(* CODESYS project device_plc_f5a.project

Project tree, tasks and I/O mapping:
  Device : C6 SMART BASIC, KEB - Karl E. Brinkmann GmbH, version 3.5.6.41
    application Application
      libraries: Standard, * (System); KEB_Gateway_Utility, * (KEB - Karl E. Brinkmann GmbH); SysTimeCore, * (System); CmpErrors, * (System); SysSocket, * (System); KEB_Drive_Utility, * (KEB - Karl E. Brinkmann GmbH); KEB_Base, * (KEB - Karl E. Brinkmann GmbH); CmpEventMgr, 3.5.5.0 (System); Component Manager, 3.5.5.0 (System); CmpApp, 3.5.6.0 (System); CmpIecTask, 3.5.5.0 (System)
      task MainTask (cyclic, interval t#4ms, priority 0) calls PLC_PRG, Gateway
      task EtherCAT_Master_C6_SMART (externalevent, external event EVENT_ECM_DC, priority 0) calls EtherCAT_Master_C6_SMART.EtherCAT_Task [EtherCAT_Master_C6_SMART.EtherCAT_Task]
      program PLC_PRG [ST]: ErrorHandling
      program MAIN [ST]
      Gateway/
        program Gateway [FBD]
        global variables GVL_GATEWAY
        global variables GVL_APP
        program SampleReadDriveParameter [FBD]
        program SampleReadMultipleParameter [ST]
        program SampleWriteDriveParameter [ST]
      SDO_RW/
        program ReadParameters [ST]
        FB/
          function block ReadPara [ST]
          function block WritePara [ST]: Dint_ToArrayOfByte
          function ArrayOfByte_to_Dword [ST]
          function block ReadParaEdge [ST]
      TCP_Server/
        function block SocketComm [ST]
        program ServerSocket [ST]: SplitRxBuffer, InitSocketFB, ComposeTxBuffer
        program PrepareStopFunction [ST]
        global variables GVL_TCP
    EtherCAT_Master_C6_SMART : EtherCAT Master C6 SMART, KEB - Karl E. Brinkmann GmbH, version 3.5.5.0
      KEB_C6_SMART_Coupler : KEB_C6_SMART_Coupler (3A E-Bus), KEB - Karl E. Brinkmann GmbH, version Revision=16#00000003
          settings: DC sync0 cycletime = 8000; DC sync1 cycletime = 8000
      KEB_F5_generic_MDP_ : KEB_F5_generic (MDP), KEB - Karl E. Brinkmann GmbH, version Revision=16#00000000
          settings: Number of Outputs = 3; Number of Inputs = 3; Number of Infos about Outputs = 3; Number of Infos about Inputs = 3; EnableExpertSettings = True; Sync.Length = 8; Sync.Length = 8; FMMU.Length = 8; FMMU.Length = 8; Number of RxPDOs of the Slave = 1; Number of TxPDOs of the Slave = 1; DC sync0 cycletime = 8000; DC enable = 1; DC sync0 enable = 1; DC sync0 factor = 'x 1'; DC sync0 shift time = 0; DC sync1 cycletime = 8000; DC sync1 enable = 0; DC sync1 factor = 'x 1'; DC sync1 shift time = 0; DCSetting = 1; RxTxPdo.NumberofExcludes = 0; RxTxPdo.NumberofEntries = 3; RxTxPdo.Index = 16#1600; RxTxPdo.Fixed = False; RxTxPdo.Mandatory = False; RxTxPdo.Virtual = False; RxTxPdo.Sm = 2; RxTxPdo.Su = 0; RxTxPdo.Name = 'Outputs'; RxTxPdo.DependOnSlot = True; RxTxPdo.DependOnSlotGroup = False; std_PD_map_F5_ PS34: ctm position [0x3322.0].Index = 16#3322; std_PD_map_F5_ PS34: ctm position [0x3322.0].SubIndex = 1; std_PD_map_F5_ PS34: ctm position [0x3322.0].Size = 32; std_PD_map_F5_ PS34: ctm position [0x3322.0].Offset = 0; std_PD_map_F5_ PS34: ctm position [0x3322.0].DependOnSlot = False; std_PD_map_F5_ PS34: ctm position [0x3322.0].DependOnSlotGroup = False; std_PD_map_F5_ Sy52: set speed value [0x2034.0].Index = 16#2034; std_PD_map_F5_ Sy52: set speed value [0x2034.0].SubIndex = 1;
            std_PD_map_F5_ Sy52: set speed value [0x2034.0].Size = 16; std_PD_map_F5_ Sy52: set speed value [0x2034.0].Offset = 0; std_PD_map_F5_ Sy52: set speed value [0x2034.0].DependOnSlot = False; std_PD_map_F5_ Sy52: set speed value [0x2034.0].DependOnSlotGroup = False; std_PD_map_F5_ Sy50: control word (low) [0x2032.0].Index = 16#2032; std_PD_map_F5_ Sy50: control word (low) [0x2032.0].SubIndex = 1; std_PD_map_F5_ Sy50: control word (low) [0x2032.0].Size = 16; std_PD_map_F5_ Sy50: control word (low) [0x2032.0].Offset = 0; std_PD_map_F5_ Sy50: control word (low) [0x2032.0].DependOnSlot = False; std_PD_map_F5_ Sy50: control word (low) [0x2032.0].DependOnSlotGroup = False; RxTxPdo.NumberofExcludes = 0; RxTxPdo.NumberofEntries = 3; RxTxPdo.Index = 16#1A00; RxTxPdo.Fixed = False; RxTxPdo.Mandatory = False; RxTxPdo.Virtual = False; RxTxPdo.Sm = 3; RxTxPdo.Su = 0; RxTxPdo.Name = 'Inputs'; RxTxPdo.DependOnSlot = True; RxTxPdo.DependOnSlotGroup = False; std_PD_map_F5_ ru54: actual position [0x2236.0].Index = 16#2236; std_PD_map_F5_ ru54: actual position [0x2236.0].SubIndex = 1; std_PD_map_F5_ ru54: actual position [0x2236.0].Size = 32; std_PD_map_F5_ ru54: actual position [0x2236.0].Offset = 0; std_PD_map_F5_ ru54: actual position [0x2236.0].DependOnSlot = False; std_PD_map_F5_ ru54: actual position [0x2236.0].DependOnSlotGroup = False; std_PD_map_F5_ Sy53: actual speed value [0x2035.0].Index = 16#2035; std_PD_map_F5_ Sy53: actual speed value [0x2035.0].SubIndex = 1; std_PD_map_F5_ Sy53: actual speed value [0x2035.0].Size = 16; std_PD_map_F5_ Sy53: actual speed value [0x2035.0].Offset = 0; std_PD_map_F5_ Sy53: actual speed value [0x2035.0].DependOnSlot = False; std_PD_map_F5_ Sy53: actual speed value [0x2035.0].DependOnSlotGroup = False; std_PD_map_F5_ Sy51: status word (low) [0x2033.0].Index = 16#2033; std_PD_map_F5_ Sy51: status word (low) [0x2033.0].SubIndex = 1; std_PD_map_F5_ Sy51: status word (low) [0x2033.0].Size = 16; std_PD_map_F5_ Sy51: status word (low) [0x2033.0].Offset = 0; std_PD_map_F5_ Sy51: status word (low) [0x2033.0].DependOnSlot = False; std_PD_map_F5_ Sy51: status word (low) [0x2033.0].DependOnSlotGroup = False; std_PD_map_F5_ PS34: ctm position [0x3322.0].Name = 'std_PD_map_F5_ PS34: ctm position [0x3322.0]';
            std_PD_map_F5_ PS34: ctm position [0x3322.0].DataType = 'DINT'; std_PD_map_F5_ PS34: ctm position [0x3322.0].Default = ''; std_PD_map_F5_ PS34: ctm position [0x3322.0].Comment = ''; std_PD_map_F5_ Sy52: set speed value [0x2034.0].Name = 'std_PD_map_F5_ Sy52: set speed value [0x2034.0]'; std_PD_map_F5_ Sy52: set speed value [0x2034.0].DataType = 'INT'; std_PD_map_F5_ Sy52: set speed value [0x2034.0].Default = ''; std_PD_map_F5_ Sy52: set speed value [0x2034.0].Comment = ''; std_PD_map_F5_ Sy50: control word (low) [0x2032.0].Name = 'std_PD_map_F5_ Sy50: control word (low) [0x2032.0]'; std_PD_map_F5_ Sy50: control word (low) [0x2032.0].DataType = 'INT'; std_PD_map_F5_ Sy50: control word (low) [0x2032.0].Default = ''; std_PD_map_F5_ Sy50: control word (low) [0x2032.0].Comment = ''; std_PD_map_F5_ ru54: actual position [0x2236.0].Name = 'std_PD_map_F5_ ru54: actual position [0x2236.0]'; std_PD_map_F5_ ru54: actual position [0x2236.0].DataType = 'DINT'; std_PD_map_F5_ ru54: actual position [0x2236.0].Default = ''; std_PD_map_F5_ ru54: actual position [0x2236.0].Comment = ''; std_PD_map_F5_ Sy53: actual speed value [0x2035.0].Name = 'std_PD_map_F5_ Sy53: actual speed value [0x2035.0]'; std_PD_map_F5_ Sy53: actual speed value [0x2035.0].DataType = 'INT'; std_PD_map_F5_ Sy53: actual speed value [0x2035.0].Default = ''; std_PD_map_F5_ Sy53: actual speed value [0x2035.0].Comment = ''; std_PD_map_F5_ Sy51: status word (low) [0x2033.0].Name = 'std_PD_map_F5_ Sy51: status word (low) [0x2033.0]'; std_PD_map_F5_ Sy51: status word (low) [0x2033.0].DataType = 'INT'; std_PD_map_F5_ Sy51: status word (low) [0x2033.0].Default = ''; std_PD_map_F5_ Sy51: status word (low) [0x2033.0].Comment = ''
          unmapped channels: std_PD_map_F5_ PS34: ctm position [0x3322.0], std_PD_map_F5_ Sy52: set speed value [0x2034.0], std_PD_map_F5_ Sy50: control word (low) [0x2032.0], std_PD_map_F5_ ru54: actual position [0x2236.0], std_PD_map_F5_ Sy53: actual speed value [0x2035.0], std_PD_map_F5_ Sy51: status word (low) [0x2033.0]
        std_PD_map_F5_ : std PD map (F5), KEB - Karl E. Brinkmann GmbH, version 0
*)

// Device/Application/Gateway/GVL_GATEWAY
{attribute 'qualified_only'} //full name must be used  to access these variables (GVL_NAME.Variable)
//Global application variables and constants
VAR_GLOBAL
	Channelhandler : KebChannelHandler; //the KEB channelhandler handles sdo communication to keb drives	
END_VAR

// Device/Application/Gateway/GVL_APP
{attribute 'qualified_only'} //full name must be used  to access these variables (GVL_NAME.Variable)
//Global application variables and constants
VAR_GLOBAL
	CycleTimeUs:ULINT; 	//Cycletime of ethercat task
	CycleTime:TIME;		//Cycletime of ethercat task

	StatusText:STRING:='Not Initialized'; //Global status text
	Error:BOOL; 	//Global error flag
	Reset:BOOL;		//Global error reset
	ResetOld:BOOL; //reset from last cycle (usage for edge detection )
END_VAR

// Device/Application/TCP_Server/GVL_TCP
VAR_GLOBAL

	TcpBufferIn : ARRAY[0..1000,0..5]OF DWORD;			// буфер частей входящей датаграммы
														// 0-я часть - параметры, которые нужно читать
	
	TcpBufferOut : ARRAY[0..1000,0..5]OF DWORD;		//буфер частей исходящей датаграммы	
	
END_VAR

// Device/Application/PLC_PRG
PROGRAM PLC_PRG
VAR
		State: INT;//application state
		
		hEvent:UDINT;
		Event_Result:UDINT;	
		firstCycleDone:BOOL;
END_VAR



//init statemachine
CASE State OF
	0://init gateway (see gateway program)
	//=============================================================================

		IF Gateway.Error THEN //check init status
			GVL_APP.StatusText := 'Error during initalization';
		ELSIF Gateway.InitDone THEN
			GVL_APP.StatusText := 'Bus Init done';
			State:= 1; //switch to next state
		ELSE
			GVL_APP.StatusText := 'Bus Init in progress';
		END_IF
	
	1: //Get cycletime of this task, save into global variable
	//=============================================================================
		
		GVL_APP.CycleTimeUs:= KEB_GetTaskCycleTimeUs();
		IF GVL_APP.CycleTimeUs> 0 THEN
			GVL_APP.CycleTime:=ULINT_TO_TIME(GVL_APP.CycleTimeUs/1000);
			State:= 2; //switch to next state
		ELSE
			GVL_APP.Error := TRUE;
			GVL_APP.StatusText := 'Invalid cycletime';
		END_IF
		
	2://init done, do main application
	//=============================================================================
		
		//SampleReadDriveParameter();		//Run IEC Slave sample for reading	 (FBD)
		//SampleReadMultipleParameter();	//Run IEC Slave sample for reading multiple parameters (ST)
		//SampleWriteDriveParameter();	//Run IEC Slave sample for writing	(ST)
		
		
		//MAIN();		//выполнение основных операций ВАРИАНТ С ПЧ
		
		
END_CASE

ErrorHandling(); //Check and reset errors


MAIN();					//выполнение основных операций ВАРИАНТ БЕЗ ПЧ

ACTION ErrorHandling:

//Check error flags
//=====================================================================
IF Gateway.Error THEN //gateway error occured
		GVL_APP.StatusText := 'Bus error';
		GVL_APP.Error:=TRUE; //set global error flag
		State:= 0;
END_IF
		
//Reset error flags
//=====================================================================	
IF GVL_APP.Reset AND GVL_APP.ResetOld=FALSE THEN //rising edge detection
	
	Gateway.Reset := TRUE; //reset gateway
	GVL_APP.Error:=FALSE; //reset global error flag
	
ELSIF GVL_APP.Reset=FALSE AND  GVL_APP.ResetOld=TRUE THEN //falling edge detection
 	
	Gateway.Reset := FALSE; //remove reset flag
	
END_IF

	
//save status for edge detection
GVL_APP.ResetOld:= GVL_APP.Reset;
END_ACTION

END_PROGRAM

// Device/Application/Gateway/Gateway
(*
	Gateway program handles sdo communication to keb drives.
	Various startup and diagnostic options are available
	
	Global variable of type KebChannelHandler is mandatory: default list and name: GVL_APP.ChannelHandler
*)

PROGRAM Gateway
VAR_INPUT
	Reset: BOOL; //reset general gateway error 
	Restart: BOOL; //restart bus 
END_VAR
VAR_OUTPUT
	InitDone:BOOL; //Gateway init done
	Error:BOOL;		//general gateway error, details see internal fbs
	ElapsedInitTime: TIME; //gateway init time
END_VAR

VAR CONSTANT
	MAX_INIT_TIME: TIME := T#120S; //max. time for initalization
END_VAR

VAR
	SetComEtc: SetCom_ETC_Master;		//the ethercat master gateway interface
	SetComDin: SetCom_DIN_Slave;		//the DIN slave for communication via COMBIVIS
	tonInitTimeout: ton;
	ResetOld: BOOL;
	EnableDin: BOOL := true;
END_VAR

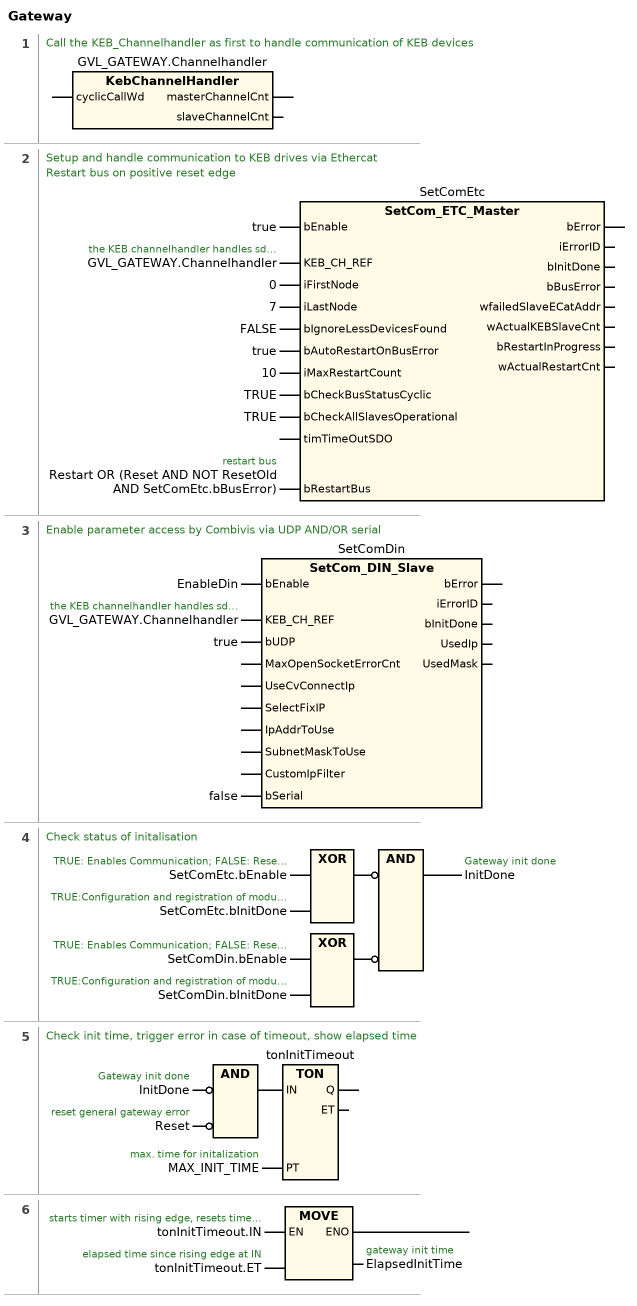
// NETWORK 1
// Call the KEB_Channelhandler as first to handle communication of KEB devices
//   GVL_GATEWAY.Channelhandler: the KEB channelhandler handles sdo communication to keb drives
GVL_GATEWAY.Channelhandler(); // KebChannelHandler

// NETWORK 2
// Setup and handle communication to KEB drives via Ethercat
// Restart bus on positive reset edge
//   SetComEtc: the ethercat master gateway interface
//   GVL_GATEWAY.Channelhandler: the KEB channelhandler handles sdo communication to keb drives
//   Restart OR (Reset AND NOT ResetOld AND SetComEtc.bBusError): restart bus
SetComEtc(
    bEnable := true,
    KEB_CH_REF := GVL_GATEWAY.Channelhandler,
    iFirstNode := 0,
    iLastNode := 7,
    bIgnoreLessDevicesFound := FALSE,
    bAutoRestartOnBusError := true,
    iMaxRestartCount := 10,
    bCheckBusStatusCyclic := TRUE,
    bCheckAllSlavesOperational := TRUE,
    bRestartBus := Restart OR (Reset AND NOT ResetOld AND SetComEtc.bBusError)); // SetCom_ETC_Master

// NETWORK 3
// Enable parameter access by Combivis via UDP AND/OR serial
//   GVL_GATEWAY.Channelhandler: the KEB channelhandler handles sdo communication to keb drives
SetComDin(bEnable := EnableDin, KEB_CH_REF := GVL_GATEWAY.Channelhandler, bUDP := true, bSerial := false); // SetCom_DIN_Slave

// NETWORK 4
// Check status of initalisation
//   SetComEtc.bEnable: TRUE: Enables Communication; FALSE: Reset FB and deregister modul. Disableing (falling edge on bEnable) is not recommended. Processed data may be lost.
//   SetComEtc.bInitDone: TRUE:Configuration and registration of modul successfully done
//   SetComDin.bEnable: TRUE: Enables Communication; FALSE: Reset FB and deregister modul. Disableing (falling edge on bEnable) is not recommended. Processed data may be lost.
//   SetComDin.bInitDone: TRUE:Configuration and registration of modul successfully done
//   InitDone: Gateway init done
InitDone := NOT (SetComEtc.bEnable XOR SetComEtc.bInitDone) AND NOT (SetComDin.bEnable XOR SetComDin.bInitDone);

// NETWORK 5
// Check init time, trigger error in case of timeout, show elapsed time
//   InitDone: Gateway init done
//   Reset: reset general gateway error
//   MAX_INIT_TIME: max. time for initalization
tonInitTimeout(IN := NOT InitDone AND NOT Reset, PT := MAX_INIT_TIME); // TON

// NETWORK 6
//   tonInitTimeout.IN: starts timer with rising edge, resets timer with falling edge
//   tonInitTimeout.ET: elapsed time since rising edge at IN
//   ElapsedInitTime: gateway init time
IF tonInitTimeout.IN THEN ElapsedInitTime := tonInitTimeout.ET; END_IF

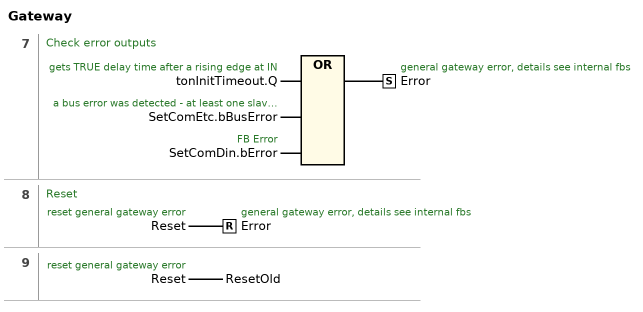
// NETWORK 7
// Check error outputs
//   tonInitTimeout.Q: gets TRUE delay time after a rising edge at IN
//   SetComEtc.bBusError: a bus error was detected - at least one slave changed its state back from operational to init.
//   SetComDin.bError: FB Error
//   Error: general gateway error, details see internal fbs
Error S= tonInitTimeout.Q OR SetComEtc.bBusError OR SetComDin.bError;

// NETWORK 8
// Reset
//   Reset: reset general gateway error
//   Error: general gateway error, details see internal fbs
Error R= Reset;

// NETWORK 9
//   Reset: reset general gateway error
ResetOld := Reset;

END_PROGRAM

// Device/Application/MAIN
PROGRAM MAIN
VAR
	
END_VAR


ServerSocket();









//test1-----------
(*
IF 1=1 THEN

read_para_3(
	StartReading:=TRUE, 
	ContinuousReading:= TRUE, 
	SlaveAddr:= KEB_F5_generic_MDP_.PhysSlaveAddr, 
	Index:= 16#2000+16#0236, 	//236-ru54 факт.позиция;    20C-ru.12 факт.момент
	SubIndex:= 16#1, 
	ReadInterval:= 200, 
	Value=> val3, 
	DoneEdge=> read_done3);
	
	//edge_detect(CLK:= read_done3, Q=> read_done );

	IF (count3<99) AND (read_done3=TRUE)  (*AND (startread=TRUE)*)  THEN
		val3_arr[count3,0]:=val3;
		val3_arr[count3,1]:=BOOL_TO_DINT(read_done3);
		val3_arr[count3,2]:=SysTimeGetMs();
		
		
		IF (count3>0) THEN
			val3_arr[count3,3]:=val3_arr[count3,2] - val3_arr[count3-1,2];
		END_IF
		
		count3:=count3+1;
	END_IF


END_IF		
		
*)		
//test1--------------

END_PROGRAM

// Device/Application/TCP_Server/ServerSocket
PROGRAM ServerSocket
VAR
											//переменные оригинальной версии Сервера
	Comm : SocketComm;
	RxBuffer : ARRAY[0..1000] OF DWORD;		//буфер приёма	15
	TxBuffer : ARRAY[0..1000] OF DWORD;		//буфер передачи	15
	inited: BOOL;
	

	
							//внедренные переменные
	count_rx	: DINT;		//счетчик элементов входящей датаграммы
	count_part	: DINT:=0;
	count_elem	: DINT:=0;

	count_zero_1	:	DINT;	//счетчик для обнуления массива частей входящй датаграммы
	count_zero_2	:	DINT;	//счетчик для обнуления массива частей входящй датаграммы	

	PrevTxCnt	:	UDINT;		//номер предыдущей отправки по ТСР
	
	count_tx_out	: DINT;		//счетчик элементов исходящей датаграммы
	count_part_out	: DINT:=0;
	count_elem_out	: DINT:=0;
	count_clean_tx	: DINT:=0;
	count_clean_rx	: DINT:=0;		
	count_clean_out	: DINT:=0;
	
	edge_detect: R_TRIG;
	time_shift : DINT;
						
	//DataLen	:	ARRAY [0..10] OF DWORD;											
	//RxBufferTemp : ARRAY[0..100] OF DWORD;	
	(*									
	counterTx	:	INT;

	arr_elem_number: INT;
	params_to_read:ARRAY[1..10] OF BOOL;
	
	read_para_1: ReadParaEdge;
	read_para_2: ReadParaEdge;
	read_para_3: ReadParaEdge;
	read_para_4: ReadParaEdge;
	
	val1:DINT;
	val2:DINT;
	val3:DINT;
	
	read_done1:BOOL;
	read_done2:BOOL;
	read_done3:BOOL;
	
	count1:INT;
	count2:INT;
	count3:INT;
	
	val1_arr:ARRAY[0..100,0..2] OF DINT;
	val2_arr:ARRAY[0..100,0..2] OF DINT;
	val3_arr:ARRAY[0..100,0..2] OF DINT;
	done_arr:ARRAY[0..100] OF BOOL;
	time_arr:ARRAY[0..100] OF dint;	
	
	del:UDINT;
	
	startread: BOOL;
	kkk: INT;	
		PrevTxCnt: UDINT;
	count_clean_tx: DINT;
	count_fill_tx: DINT;
	
	
	j:int;
	*)
END_VAR

InitSocketFB();		//Инициализация параметров функционального блока сокета




Comm();				//вызов ФБ сокета



IF Comm.PartnerIp = '' THEN
	FOR count_clean_rx:=0 TO 1000 DO				//обнуление входящей датаграммы
		RxBuffer[count_clean_rx] :=0;
	END_FOR
END_IF

SplitRxBuffer();	//распределение датаграммы на составные части и включение их в буфер GVL_TCP.TcpBufferIn



edge_detect(CLK:= ( Comm.PartnerIp <> '' ), Q=>  );
IF edge_detect.Q=TRUE THEN time_shift:= SysTimeGetMs(); END_IF
ReadParameters();	//чтение параметров через SDO




//если только что была сделана отправка (см. "старый код") то вызываем ComposeTxBuffer
// Он собирает TxBuffer из частей датаграммы отправки, а сами части чистит
IF ServerSocket.Comm.TxCnt > PrevTxCnt THEN							//если произошла отправка буфера по ТСР
	ComposeTxBuffer();												//вызываем сборку исходящей датаграммы из частей
	Comm.TxLen:= DWORD_TO_INT(TxBuffer[0] + 1) * 4;			//устанавливаем кол-во байт для передачи
	PrevTxCnt:=ServerSocket.Comm.TxCnt;
END_IF

IF Comm.PartnerIp = '' THEN
	FOR count_clean_tx:=0 TO 1000 DO				//обнуление исходящей датаграммы
		TxBuffer[count_clean_tx] :=0;
	END_FOR
	Comm.TxLen:= DWORD_TO_INT(TxBuffer[0] + 1) * 4;
END_IF




(*																	//очистка буфера отправки по нарастающему фронту количества отправок
IF ServerSocket.Comm.TxCnt > PrevTxCnt THEN							//если произошла отправка буфера по ТСР
	FOR count_clean_tx:=0 TO SIZEOF(ServerSocket.TxBuffer)/4 DO
		ServerSocket.TxBuffer[count_clean_tx]:=0;
		count_fill_tx:=0;
	END_FOR
	PrevTxCnt:=ServerSocket.Comm.TxCnt;
END_IF
*)




(*
read_para_1(					//-----
	StartReading:=TRUE, 
	ContinuousReading:= TRUE, 
	SlaveAddr:= KEB_F5_generic_MDP_.PhysSlaveAddr, 
	Index:= 16#2000+16#0236, 	//-----//236-ru54 факт.позиция;    20C-ru.12 факт.момент;		20F-ru.15 полный ток
	SubIndex:= 16#1, 
	ReadInterval:= 200, 
	Value=> , 
	DoneEdge=> );
IF read_para_1.DoneEdge=TRUE  THEN									//-----		
	ServerSocket.TxBuffer[count_fill_tx+1]:=1;						//-----
	ServerSocket.TxBuffer[count_fill_tx+2]:=read_para_1.Value;		//-----			
	ServerSocket.TxBuffer[count_fill_tx+3]:=SysTimeGetMs();
	
	count_fill_tx:=count_fill_tx+3;
	ServerSocket.TxBuffer[0]:=ServerSocket.TxBuffer[0]+3;
END_IF


read_para_2(					//-----
	StartReading:=TRUE, 
	ContinuousReading:= TRUE, 
	SlaveAddr:= KEB_F5_generic_MDP_.PhysSlaveAddr, 
	Index:= 16#2000+16#020C, 	//-----//236-ru54 факт.позиция;    20C-ru.12 факт.момент;		20F-ru.15 полный ток
	SubIndex:= 16#1, 
	ReadInterval:= 300, 
	Value=> , 
	DoneEdge=> );
IF read_para_2.DoneEdge=TRUE  THEN									//-----		
	ServerSocket.TxBuffer[count_fill_tx+1]:=2;						//-----
	ServerSocket.TxBuffer[count_fill_tx+2]:=read_para_2.Value;		//-----			
	ServerSocket.TxBuffer[count_fill_tx+3]:=SysTimeGetMs();
	
	count_fill_tx:=count_fill_tx+3;
	ServerSocket.TxBuffer[0]:=ServerSocket.TxBuffer[0]+3;
END_IF


read_para_3(					//-----
	StartReading:=TRUE, 
	ContinuousReading:= TRUE, 
	SlaveAddr:= KEB_F5_generic_MDP_.PhysSlaveAddr, 
	Index:= 16#2000+16#020F, 	//-----//236-ru54 факт.позиция;    20C-ru.12 факт.момент;		20F-ru.15 полный ток
	SubIndex:= 16#1, 
	ReadInterval:= 300, 
	Value=> , 
	DoneEdge=> );
IF read_para_3.DoneEdge=TRUE  THEN									//-----		
	ServerSocket.TxBuffer[count_fill_tx+1]:=3;						//-----
	ServerSocket.TxBuffer[count_fill_tx+2]:=read_para_3.Value;		//-----			
	ServerSocket.TxBuffer[count_fill_tx+3]:=SysTimeGetMs();
	
	count_fill_tx:=count_fill_tx+3;
	ServerSocket.TxBuffer[0]:=ServerSocket.TxBuffer[0]+3;
END_IF


read_para_4(					//-----
	StartReading:=TRUE, 
	ContinuousReading:= TRUE, 
	SlaveAddr:= KEB_F5_generic_MDP_.PhysSlaveAddr, 
	Index:= 16#2000+16#0200, 	//-----//236-ru54 факт.позиция;    20C-ru.12 факт.момент;		20F-ru.15 полный ток
	SubIndex:= 16#1, 
	ReadInterval:= 90, 
	Value=> , 
	DoneEdge=> );
IF read_para_4.DoneEdge=TRUE  THEN									//-----		
	ServerSocket.TxBuffer[count_fill_tx+1]:=4;						//-----
	ServerSocket.TxBuffer[count_fill_tx+2]:=read_para_4.Value;		//-----			
	ServerSocket.TxBuffer[count_fill_tx+3]:=SysTimeGetMs();
	
	count_fill_tx:=count_fill_tx+3;
	ServerSocket.TxBuffer[0]:=ServerSocket.TxBuffer[0]+3;
END_IF
*)



//Comm.TxLen:= DWORD_TO_INT(   TxBuffer[0]+1    ) * 4;



























//-----------------------------------старый код----------------------------------------------





	//FOR count_rx:=1 TO DWORD_TO_DINT(RxBuffer[0]) DO	//отсчет элементов дейтаграммы, не считая 1й (общая длина)
	//	IF part_now=FALSE THEN 
	//END_FOR												//count_rx:=1 TO RxBuffer[0] DO











(*	//DataLen[0]:=RxBuffer[0];
	//DataLen[1]:=RxBuffer[1];
	FOR i:=0 TO 100 DO 
		IF (i MOD 2)=0 THEN j:=0; ELSE j:=1; END_IF
		IF i=0 THEN j:=0; END_IF
		
		RxBufferTemp[i]:=RxBuffer[j];
	END_FOR
	*)






(*
IF params_to_read[1]=TRUE THEN
	read_para_1(
		StartReading:=TRUE, 
		ContinuousReading:= TRUE, 
		SlaveAddr:= KEB_F5_generic_MDP_.PhysSlaveAddr, 
		Index:= 16#2000+16#0200, 	//236-ru54 факт.позиция;    20C-ru.12 факт.момент
		SubIndex:= 16#1, 
		ReadInterval:= 200, 
		Value=> val1, 
		Done=> read_done1);	
END_IF
*)




(*	
IF params_to_read[2]=TRUE THEN

read_para_2(
	StartReading:=TRUE, 
	ContinuousReading:= TRUE,//TRUE, 
	SlaveAddr:= KEB_F5_generic_MDP_.PhysSlaveAddr, 
	Index:= 16#2000+16#0207, 	//236-ru54 факт.позиция;    20C-ru.12 факт.момент
	SubIndex:= 16#1, 
	ReadInterval:= 200, 
	Value=> val2, 
	DoneEdge=> read_done2);

//IF 1=1 THEN														//вариант без ПЧ
IF (read_done2=TRUE) (*AND (startread=TRUE)*)  THEN			//вариант с ПЧ
	
	ServerSocket.TxBuffer[count_fill_tx+1]:=2;
	
	//ServerSocket.TxBuffer[count_fill_tx+2]:=136;				//вариант без ПЧ
	ServerSocket.TxBuffer[count_fill_tx+2]:=val2;				//вариант с ПЧ
	
	ServerSocket.TxBuffer[count_fill_tx+3]:=SysTimeGetMs();
	
	count_fill_tx:=count_fill_tx+3;
	ServerSocket.TxBuffer[0]:=ServerSocket.TxBuffer[0]+3;
END_IF	
END_IF	







IF params_to_read[3]=TRUE THEN

read_para_3(
	StartReading:=TRUE, 
	ContinuousReading:= TRUE, 
	SlaveAddr:= KEB_F5_generic_MDP_.PhysSlaveAddr, 
	Index:= 16#2000+16#020C, 	//236-ru54 факт.позиция;    20C-ru.12 факт.момент
	SubIndex:= 16#1, 
	ReadInterval:= 200, 
	Value=> val3, 
	DoneEdge=> read_done3);


//IF 1=1 THEN														//вариант без ПЧ
IF (read_done3=TRUE) (*AND (startread=TRUE)*)  THEN			//вариант с ПЧ

	ServerSocket.TxBuffer[count_fill_tx+1]:=3;
	
	//ServerSocket.TxBuffer[count_fill_tx+2]:=288;				//вариант без ПЧ
	ServerSocket.TxBuffer[count_fill_tx+2]:=val3;				//вариант с ПЧ
	
	ServerSocket.TxBuffer[count_fill_tx+3]:=SysTimeGetMs();
	
	count_fill_tx:=count_fill_tx+3;
	ServerSocket.TxBuffer[0]:=ServerSocket.TxBuffer[0]+3;

END_IF
END_IF	






//4 param
IF params_to_read[3]=TRUE THEN

read_para_4(
	StartReading:=TRUE, 
	ContinuousReading:= TRUE, 
	SlaveAddr:= KEB_F5_generic_MDP_.PhysSlaveAddr, 
	Index:= 16#2000+16#020F, 	//236-ru54 факт.позиция;    20C-ru.12 факт.момент;		20F-ru.15 полный ток
	SubIndex:= 16#1, 
	ReadInterval:= 200, 
	Value=> , 
	DoneEdge=> );


IF (read_para_4.DoneEdge=TRUE) (*AND (startread=TRUE)*)  THEN			

	ServerSocket.TxBuffer[count_fill_tx+1]:=4;
	
	ServerSocket.TxBuffer[count_fill_tx+2]:=read_para_4.Value;				
	
	ServerSocket.TxBuffer[count_fill_tx+3]:=SysTimeGetMs();
	
	count_fill_tx:=count_fill_tx+3;
	ServerSocket.TxBuffer[0]:=ServerSocket.TxBuffer[0]+3;

END_IF
END_IF	
*)












(*IF NOT firstCycleDone THEN
	hEvent:=EventOpen(EVT_Logout, CMPID_CmpApp, Event_Result);
	Event_Result:=EventRegisterCallbackFunction(hEvent, ADR(PrepareStopFunction));
	firstCycleDone:=TRUE;
END_IF*)
//EventIDs.EVT_PrepareStop















//------------------захват переметров-------------------------
(*
FOR arr_elem_number:=1 TO 10 DO												//обнуление  массива номеров параметров, которые необходимо читать
	params_to_read[arr_elem_number]:=FALSE;
END_FOR


FOR arr_elem_number:=1 TO DWORD_TO_INT(ServerSocket.RxBuffer[0]) DO			//заполнение массива номеров параметров, которые необходимо читать
	IF ServerSocket.RxBuffer[arr_elem_number]>0 THEN
		params_to_read[ServerSocket.RxBuffer[arr_elem_number] ]:= TRUE;
		
	END_IF
END_FOR
*)












(*
IF (count1<100) AND (read_done1=TRUE) AND (startread=TRUE)  THEN
	val1_arr[count1,0]:=val2;
	val1_arr[count1,1]:=BOOL_TO_DINT(read_done2);
	val1_arr[count1,2]:=SysTimeGetMs();
	count1:=count1+1;
END_IF


IF (count2<100) AND (read_done2=TRUE) AND (startread=TRUE)  THEN
	val2_arr[count2,0]:=val2;
	val2_arr[count2,1]:=BOOL_TO_DINT(read_done2);
	val2_arr[count2,2]:=SysTimeGetMs();
	count2:=count2+1;
END_IF


IF (count3<100) AND (read_done3=TRUE)  AND (startread=TRUE)  THEN
	val3_arr[count3,0]:=val3;
	val3_arr[count3,1]:=BOOL_TO_DINT(read_done3);
	val3_arr[count3,2]:=SysTimeGetMs();
		count3:=count3+1;
END_IF
*)











//TxBuffer[0] := 3*SIZEOF(TxBuffer[0]);
//TxBuffer[1] := 2;
//TxBuffer[2] := 5;
//TxBuffer[3] := 7;

(*TxBuffer[0] := 0;											//предварительное обнуление заголовка длины дейтаграммы
counterTx:=1;												//счетчик элементов дейтаграммы устанавливается равным 1, т.к. по умолчанию всегда есть как минимум 1 элемент - заголовок длины
WHILE (TxBuffer[counterTx] <>0) DO
	counterTx:=counterTx+1;									//если очередной элемент буфера отправки ненулевой, то счетчик увеличивается
END_WHILE
TxBuffer[0]:=counterTx-1;
Comm.TxLen:=counterTx*SIZEOF(TxBuffer[0]);
*)

ACTION SplitRxBuffer:
//распределение датаграммы на составные части и включение их в буфер GVL_TCP.TcpBufferIn


IF Comm.PartnerIp <>'' THEN											//если есть входящее подключение
	count_rx:=1;													//сброс: счетчик элементов датаграммы на 1 (отсчет всех элементов не считая "общей длины датаграммы"
	count_part:=0;													//		 счетчика частей датаграммы
	count_elem:=0;													//		 счетчика элементов частей

	WHILE count_rx <= RxBuffer[0] DO								//пока не прочитаны все элементы дагараммы
		GVL_TCP.TcpBufferIn[count_elem, count_part] := RxBuffer[count_rx];	//добавляем к ТСРБуферу текущий элемент датаграммы
		IF count_elem >= TcpBufferIn[0, count_part] THEN				//если считаны все элементы текущей части (если номер "элемента части датаграммы" не более "длины части")
			count_part := count_part + 1;							//увеличиваем счетчик частей
			count_elem := 0;										//обнуляем счетчик элементов части
		ELSE
			count_elem := count_elem + 1;							//увеличиваем счетчик элементов части
		END_IF
		count_rx := count_rx + 1;									//увеличиваем счетчик элементов датаграммы
	END_WHILE
ELSE

	FOR count_zero_1:=0 TO 1000 DO									//если нет подключения по ТСР - обнуляем все части входящей датаграммы
		FOR count_zero_2:=0 TO 5 DO	
			GVL_TCP.TcpBufferIn[count_zero_1, count_zero_2]:=0;
		END_FOR
	END_FOR
END_IF													//IF Comm.PartnerIp <>'' THEN
END_ACTION

ACTION InitSocketFB:

IF NOT inited THEN							
	inited := TRUE;
	Comm.Host := '';						//wait for incoming requests from any partner
	Comm.UseTcp := TRUE;					//Use TCP
	Comm.pRxBuffer := ADR(RxBuffer);
	Comm.MaxRxLen := SIZEOF(RxBuffer);		//receive as long as our buffer can hold data
	Comm.pTxBuffer := ADR(TxBuffer);		
	Comm.TxLen := 4;	//0;	//200;//24;					//transmit 24 bytes only
	Comm.Enable := TRUE;					//start immediately
ELSE
	//Comm.Enable := NOT (PrepareStopFunction.DelSockets);	
END_IF
END_ACTION

ACTION ComposeTxBuffer:
FOR count_clean_tx:=0 TO 1000 DO				//обнуление исходящей датаграммы
	TxBuffer[count_clean_tx] :=0;
END_FOR



	
	count_tx_out:=1;								//сброс счетчика элементов исходящей датаграммыж на 1й элемент (0й - общая длина датаграммы)
	
																							//соединение составных частей (GVL_TCP.TcpBufferIn) в исходящую датаграмму 
	FOR count_part_out:=0 TO 5 DO															//перебор частей датаграммы
		FOR count_elem_out:=0 TO TcpBufferOut[0 ,count_part_out] DO							//перебор элементов частей дагарммы
			IF count_elem_out=0 THEN
				TxBuffer[0] := TxBuffer[0] + TcpBufferOut[count_elem_out, count_part_out] + 1;	//если текущий элемент - первый в части, то он - длина части и его значение (+1 для учета самогО элемента) прибавляется к общей длине исходящей датаграммы 
			END_IF
			
			TxBuffer[count_tx_out] := TcpBufferOut[count_elem_out, count_part_out];			//присвоение очередному элементу исходящей датаграммы значения текущего элемента текущей части
			count_tx_out := count_tx_out + 1;
			
			//TcpBufferOut[count_elem_out, count_part_out] := 0;								//обнуление элемента части исходящей датаграммы
		
		END_FOR
	END_FOR
	
	
	FOR count_part_out:=0 TO 5 DO								//перебор частей датаграммы
		FOR count_elem_out:=0 TO 1000 DO						//перебор элементов частей дагарммы
			TcpBufferOut[count_elem_out, count_part_out] := 0;								//обнуление элемента части исходящей датаграммы
		END_FOR
	END_FOR	
	

	
	
(*

	count_rx_out	: DINT;		//счетчик элементов исходящей датаграммы
	count_part_out	: DINT:=0;
	count_elem_out	: DINT:=0;

*)
END_ACTION

END_PROGRAM

// Device/Application/SDO_RW/ReadParameters
PROGRAM ReadParameters
VAR
	counter: DINT;								//чсетчик цикла обнуления массива номеров параметров, которые необходимо прочитать
	paramsToRead:ARRAY[1..1000] OF BOOL;		

	time_interval	:	DINT;					//интервал считвания параметров по SDO
	counter_fill	:	DINT;
	read_para_1,	
	read_para_2,	
	read_para_3,	
	read_para_4	
					:	ReadParaEdge;	

	counter_zero	:	DINT;
END_VAR

IF  (GVL_TCP.TcpBufferIn[0, 0] > 0) AND (GVL_TCP.TcpBufferIn[0, 0] < 1000) THEN	//параметры считываются только при корректной входящей датаграмме
	

	FOR counter:=1 TO 1000 DO
		paramsToRead[counter]:=FALSE;									//обнуление  массива номеров параметров, которые необходимо читать
	END_FOR
	
	
	FOR counter:=1 TO TcpBufferIn[0,0] DO
		IF GVL_TCP.TcpBufferIn[counter, 0] > 0 THEN
			paramsToRead[ GVL_TCP.TcpBufferIn[counter, 0] ] := TRUE;	//заполнение  массива номеров параметров, которые необходимо читать
		END_IF
	END_FOR
	
	
	time_interval:= GVL_TCP.TcpBufferIn[0, 0]*100;						//установка интервала считывания параметров (по 100 мс на каждый параметр)



	
	IF GVL_TCP.TcpBufferOut[0,0] < 900 THEN			//если часть отправляемой датаграммы еще не переполнена
		// 1
		IF paramsToRead[1]=TRUE THEN											//-----
			read_para_1(														//-----
				StartReading:=TRUE, 
				ContinuousReading:= TRUE, 
				SlaveAddr:= KEB_F5_generic_MDP_.PhysSlaveAddr, 
				Index:= 16#2000+16#0200, 										//-----//236-ru54 факт.позиция;    20C-ru.12 факт.момент;		20F-ru.15 полный ток
				SubIndex:= 16#1, 
				ReadInterval:= time_interval, 
				Value=> , 
				DoneEdge=> );
			//IF 1=1 THEN
			IF read_para_1.DoneEdge=TRUE  THEN									//-----		
				counter_fill := GVL_TCP.TcpBufferOut[0,0];
				GVL_TCP.TcpBufferOut[counter_fill+1, 0] := 1;					//-----
				GVL_TCP.TcpBufferOut[counter_fill+2, 0] :=read_para_1.Value;	//-----			
				GVL_TCP.TcpBufferOut[counter_fill+3, 0] :=SysTimeGetMs() - ServerSocket.time_shift;
				GVL_TCP.TcpBufferOut[0,0] := GVL_TCP.TcpBufferOut[0,0] + 3;
			END_IF
		END_IF

		// 2
		IF paramsToRead[2]=TRUE THEN											//-----
			read_para_2(														//-----
				StartReading:=TRUE, 
				ContinuousReading:= TRUE, 
				SlaveAddr:= KEB_F5_generic_MDP_.PhysSlaveAddr, 
				Index:= 16#2000+16#0035, 										//-- ?/16#0207---//236-ru54 факт.позиция;    20C-ru.12 факт.момент;		20F-ru.15 полный ток
				SubIndex:= 16#1, 
				ReadInterval:= time_interval, 
				Value=> , 
				DoneEdge=> );
			//IF 1=1 THEN
			IF read_para_2.DoneEdge=TRUE  THEN									//-----		
				counter_fill := GVL_TCP.TcpBufferOut[0,0];
				GVL_TCP.TcpBufferOut[counter_fill+1, 0] := 2;					//-----
				GVL_TCP.TcpBufferOut[counter_fill+2, 0] := DINT_TO_INT(read_para_2.Value);  //read_para_2.Value;	//-----			
				GVL_TCP.TcpBufferOut[counter_fill+3, 0] :=SysTimeGetMs()  - ServerSocket.time_shift;
				GVL_TCP.TcpBufferOut[0,0] := GVL_TCP.TcpBufferOut[0,0] + 3;
			END_IF
		END_IF		
		
		
		IF paramsToRead[3]=TRUE THEN											//-----
			read_para_3(														//-----
				StartReading:=TRUE, 
				ContinuousReading:= TRUE, 
				SlaveAddr:= KEB_F5_generic_MDP_.PhysSlaveAddr, 
				Index:= 16#2000+16#020C, 										//-----//236-ru54 факт.позиция;    20C-ru.12 факт.момент;		20F-ru.15 полный ток
				SubIndex:= 16#1, 
				ReadInterval:= time_interval, 
				Value=> , 
				DoneEdge=> );
			//IF 1=1 THEN	
			IF read_para_3.DoneEdge=TRUE  THEN									//-----		
				counter_fill := GVL_TCP.TcpBufferOut[0,0];
				GVL_TCP.TcpBufferOut[counter_fill+1, 0] := 3;					//-----
				GVL_TCP.TcpBufferOut[counter_fill+2, 0] := read_para_3.Value;	//-----			
				GVL_TCP.TcpBufferOut[counter_fill+3, 0] :=SysTimeGetMs()  - ServerSocket.time_shift;
				GVL_TCP.TcpBufferOut[0,0] := GVL_TCP.TcpBufferOut[0,0] + 3;
			END_IF
		END_IF	


		
		IF paramsToRead[4]=TRUE THEN											//-----
			read_para_4(														//-----
				StartReading:=TRUE, 
				ContinuousReading:= TRUE, 
				SlaveAddr:= KEB_F5_generic_MDP_.PhysSlaveAddr, 
				Index:= 16#2000+16#0236, 										//-----//236-ru54 факт.позиция;    20C-ru.12 факт.момент;		20F-ru.15 полный ток
				SubIndex:= 16#1, 
				ReadInterval:= time_interval, 
				Value=> , 
				DoneEdge=> );
			//IF 1=1 THEN	
			IF read_para_4.DoneEdge=TRUE  THEN									//-----		
				counter_fill := GVL_TCP.TcpBufferOut[0,0];
				GVL_TCP.TcpBufferOut[counter_fill+1, 0] := 4;					//-----
				GVL_TCP.TcpBufferOut[counter_fill+2, 0] := read_para_4.Value;	//-----			
				GVL_TCP.TcpBufferOut[counter_fill+3, 0] :=SysTimeGetMs() - ServerSocket.time_shift;
				GVL_TCP.TcpBufferOut[0,0] := GVL_TCP.TcpBufferOut[0,0] + 3;
			END_IF
		END_IF
		
		
	END_IF

	
		(*	
		read_para_2(					//-----
			StartReading:=TRUE, 
			ContinuousReading:= TRUE, 
			SlaveAddr:= KEB_F5_generic_MDP_.PhysSlaveAddr, 
			Index:= 16#2000+16#0207, 	//-----//236-ru54 факт.позиция;    20C-ru.12 факт.момент;		20F-ru.15 полный ток
			SubIndex:= 16#1, 
			ReadInterval:= 300, 
			Value=> , 
			DoneEdge=> );
		IF read_para_2.DoneEdge=TRUE  THEN									//-----		
			ServerSocket.TxBuffer[counter_fill+1]:=2;						//-----
			ServerSocket.TxBuffer[counter_fill+2]:=read_para_2.Value;		//-----			
			ServerSocket.TxBuffer[counter_fill+3]:=SysTimeGetMs();
			
			counter_fill:=counter_fill+3;
			ServerSocket.TxBuffer[0]:=ServerSocket.TxBuffer[0]+3;
		END_IF
		
		
		read_para_3(					//-----
			StartReading:=TRUE, 
			ContinuousReading:= TRUE, 
			SlaveAddr:= KEB_F5_generic_MDP_.PhysSlaveAddr, 
			Index:= 16#2000+16#020C, 	//-----//236-ru54 факт.позиция;    20C-ru.12 факт.момент;		20F-ru.15 полный ток
			SubIndex:= 16#1, 
			ReadInterval:= 300, 
			Value=> , 
			DoneEdge=> );
		IF read_para_3.DoneEdge=TRUE  THEN									//-----		
			ServerSocket.TxBuffer[counter_fill+1]:=3;						//-----
			ServerSocket.TxBuffer[counter_fill+2]:=read_para_3.Value;		//-----			
			ServerSocket.TxBuffer[counter_fill+3]:=SysTimeGetMs();
			
			counter_fill:=counter_fill+3;
			ServerSocket.TxBuffer[0]:=ServerSocket.TxBuffer[0]+3;
		END_IF
		
	
		read_para_4(					//-----
			StartReading:=TRUE, 
			ContinuousReading:= TRUE, 
			SlaveAddr:= KEB_F5_generic_MDP_.PhysSlaveAddr, 
			Index:= 16#2000+16#0200, 	//-----//236-ru54 факт.позиция;    20C-ru.12 факт.момент;		20F-ru.15 полный ток
			SubIndex:= 16#1, 
			ReadInterval:= 90, 
			Value=> , 
			DoneEdge=> );
		IF read_para_4.DoneEdge=TRUE  THEN									//-----		
			ServerSocket.TxBuffer[count_fill_tx+1]:=4;						//-----
			ServerSocket.TxBuffer[count_fill_tx+2]:=read_para_4.Value;		//-----			
			ServerSocket.TxBuffer[count_fill_tx+3]:=SysTimeGetMs();
			
			count_fill_tx:=count_fill_tx+3;
			ServerSocket.TxBuffer[0]:=ServerSocket.TxBuffer[0]+3;
		END_IF
		*)
	
	
//END_IF		//IF GVL_TCP.TcpBufferOut[0,0] < 900 THEN			//если часть отправляемой датаграммы еще не переполнена	
	
	
	//Comm.TxLen:= DWORD_TO_INT(   TxBuffer[0]+1    ) * 4;

	
ELSE												//если пришла некоректная и нулевая входная датаграмма
	FOR counter_zero:=0 TO 1000 DO					//обнуление части исходящей датограммы со считанными параметрами
		GVL_TCP.TcpBufferOut[counter_zero, 0] := 0;
	END_FOR
END_IF		//IF  GVL_TCP.TcpBufferIn[0, 0] > 0 AND GVL_TCP.TcpBufferIn[0, 0] < 1000	//параметры считываются только при корректной входящей датаграмме










//------------------захват переметров-------------------------
(*
FOR arr_elem_number:=1 TO 10 DO												//обнуление  массива номеров параметров, которые необходимо читать
	params_to_read[arr_elem_number]:=FALSE;
END_FOR


FOR arr_elem_number:=1 TO DWORD_TO_INT(ServerSocket.RxBuffer[0]) DO			//заполнение массива номеров параметров, которые необходимо читать
	IF ServerSocket.RxBuffer[arr_elem_number]>0 THEN
		params_to_read[ServerSocket.RxBuffer[arr_elem_number] ]:= TRUE;
		
	END_IF
END_FOR
*)

END_PROGRAM

// Device/Application/SDO_RW/FB/ReadParaEdge
FUNCTION_BLOCK ReadParaEdge
VAR_INPUT
	StartReading: BOOL;			//TRUE 		на время чтения
	ContinuousReading: BOOL;	//TRUE 		чтобы постоянно шло чтение параметра
	SlaveAddr: UINT;			//KEB_F5_generic_MDP_.PhysSlaveAddr		(похоже - это адрес EtherCAT)
	Index: WORD;				//16#2236			адрес параметра с прибавлением 2000. В этом примере это ru.54)
	SubIndex: BYTE;				//16#1				субиндекс (вроде бы везде 1)
	ReadInterval: DINT;			//200				в КЕБе ставят 200мс
END_VAR
VAR_OUTPUT
	Value: DINT;
	Done: BOOL;
	DoneEdge:BOOL;		//добавлено
END_VAR
VAR
	EC_COE_Read:  ETC_CO_SdoRead4;
	Busy, Reading_Err: BOOL;
	Execute: BOOL;
	Busy_Fall: F_TRIG;
	Reading_Step: INT;
	Value_internal: ARRAY [1..4] OF BYTE; 
	T_Out: TON;
	ReadIntervalTimer: TON;
	//Val: DINT;
	//nnn: DINT;
	mmm: DINT;
	
	edge_detect: R_TRIG; 		//добавлено
END_VAR

IF StartReading THEN
CASE Reading_Step OF
	0://Init
	
	EC_COE_Read.usiCom:= 1; 
	EC_COE_Read.uiDevice:= SlaveAddr;  
	EC_COE_Read.wIndex:= Index; 
	EC_COE_Read.bySubindex:= SubIndex; 
	EC_COE_Read.udiTimeOut:= 1000; 
	//EC_COE_Read(xExecute:= FALSE, xAbort := FALSE);
	Reading_Step := Reading_Step + 1; 
	
	1://Call untill falling edge bBusy or bError
		EC_COE_Read(xExecute:= TRUE,xAbort := FALSE, abyData => Value_internal); 
	
		//Watchdog timer	
		IF NOT Done THEN
			T_Out(IN:= TRUE, PT:= T#500MS);
		END_IF;
			
		IF EC_COE_Read.xDone AND NOT EC_COE_Read.xError THEN//Copy data to output value
			Done := TRUE;
			//mmm := mmm + 1;
			Value_internal := EC_COE_Read.abyData; 
			Value := DWORD_TO_DINT(ArrayOfByte_to_Dword(Data := Value_Internal));
			T_Out(IN:= FALSE, PT:= T#500MS);//Reset watchdog
		END_IF
		
		IF EC_COE_Read.xError OR T_Out.Q THEN//In case of watchdog or error go to reset
			Reading_Step := 2;
			T_Out(IN:= FALSE, PT:= T#500MS);
		END_IF;

		ReadIntervalTimer(IN:= ContinuousReading, PT:= DINT_TO_TIME(ReadInterval));
		IF ContinuousReading AND ReadIntervalTimer.Q THEN//reading was succesfull, after reading pause go to reset
			ReadIntervalTimer(IN:= FALSE, PT:= DINT_TO_TIME(ReadInterval));
			Reading_Step := 2;
		END_IF; 
		
	2://Reset FB
		
			EC_COE_Read(xExecute:= FALSE, xAbort := TRUE);
			Done := FALSE;
			Reading_Step := 0;
		
END_CASE
ELSE
	EC_COE_Read(xExecute:= FALSE, xAbort := FALSE);
	Done := FALSE;
	Reading_Step := 0;
END_IF

edge_detect(CLK:= Done, Q=> DoneEdge );

END_FUNCTION_BLOCK

// Device/Application/SDO_RW/FB/ArrayOfByte_to_Dword
FUNCTION ArrayOfByte_to_Dword : Dword
VAR_INPUT
	Data: ARRAY [1..4] OF BYTE;
END_VAR
VAR
END_VAR


ArrayOfByte_to_Dword.0 := Data[1].0;

ArrayOfByte_to_Dword.1 := Data[1].1;

ArrayOfByte_to_Dword.2 := Data[1].2;

ArrayOfByte_to_Dword.3 := Data[1].3;

ArrayOfByte_to_Dword.4 := Data[1].4;

ArrayOfByte_to_Dword.5 := Data[1].5;

ArrayOfByte_to_Dword.6 := Data[1].6;

ArrayOfByte_to_Dword.7 := Data[1].7;

ArrayOfByte_to_Dword.8 := Data[2].0;

ArrayOfByte_to_Dword.9 := Data[2].1;

ArrayOfByte_to_Dword.10 := Data[2].2;

ArrayOfByte_to_Dword.11 := Data[2].3;

ArrayOfByte_to_Dword.12 := Data[2].4;

ArrayOfByte_to_Dword.13 := Data[2].5;

ArrayOfByte_to_Dword.14 := Data[2].6;

ArrayOfByte_to_Dword.15 := Data[2].7;

ArrayOfByte_to_Dword.16 := Data[3].0;

ArrayOfByte_to_Dword.17 := Data[3].1;

ArrayOfByte_to_Dword.18 := Data[3].2;

ArrayOfByte_to_Dword.19 := Data[3].3;

ArrayOfByte_to_Dword.20 := Data[3].4;

ArrayOfByte_to_Dword.21 := Data[3].5;

ArrayOfByte_to_Dword.22 := Data[3].6;

ArrayOfByte_to_Dword.23 := Data[3].7;

ArrayOfByte_to_Dword.24 := Data[4].0;

ArrayOfByte_to_Dword.25 := Data[4].1;

ArrayOfByte_to_Dword.26 := Data[4].2;

ArrayOfByte_to_Dword.27 := Data[4].3;

ArrayOfByte_to_Dword.28 := Data[4].4;

ArrayOfByte_to_Dword.29 := Data[4].5;

ArrayOfByte_to_Dword.30 := Data[4].6;

ArrayOfByte_to_Dword.31 := Data[4].7;

END_FUNCTION

// Device/Application/TCP_Server/PrepareStopFunction
PROGRAM PrepareStopFunction
VAR //RETAIN
	DelSockets: BOOL;
END_VAR

//DelSockets:=TRUE;

END_PROGRAM

// Device/Application/TCP_Server/SocketComm
(* Sample TCP and UDP socket communication block. <br> 
Client starts connection and sends data, <br>
server receives and sends back own data.
*)
FUNCTION_BLOCK SocketComm
VAR_INPUT
	Enable : BOOL;							//TRUE enables operation, FALSE closes all sockets
	pTxBuffer : POINTER TO BYTE;			//Start of transmitted data
	pRxBuffer : POINTER TO BYTE;			//Start of received data
	MaxRxLen : INT;							//maximum buffer length for receiving
	TxLen : INT;							//number of bytes to transmit
	UseTcp : BOOL;							//Use TCP or default = UDP	
	Host : STRING ;							//client = ip address of remote partner, server = empty
	Port : WORD := 8013;					//used IP port. Must be the same on both partners.	8010
	RxTimeout : TIME := T#300S;				//time before closing socket without new data
END_VAR
VAR_OUTPUT
	PartnerIp : STRING;						//Ip address of partner
	NewConnections, ClosedCnt: UDINT;
	TxCnt,RxCnt,TimeoutCnt : UDINT;
END_VAR
VAR
	step : INT;
  	hdl,wrk,tmp : POINTER TO BYTE :=  SysTypes.RTS_INVALID_HANDLE;	
	OS : OpenSocket;						//Socket opening fb from KebBase lib
	SH : SocketHandling;					//Socket handling fb from KebBase lib
	Tout : ton;
	result: UDINT;
	di,cnt : DINT;
	WaitForRsp: BOOL;
//------	
	ManualClose:BOOL;	//добавленная переменная - ручное отключение сервера
	stateString:STRING;
	
	
	
END_VAR


CASE step OF
	0:
	  IF Enable THEN
		  IF pTxBuffer = 0 OR pRxBuffer = 0 THEN
			  Step := 200;									//error - no buffers assigned
			  RETURN;
		  END_IF
		  Step := step + 1;
	  END_IF
	  
	1:	//create socket
		SH.Tcp := UseTcp;									//select between TCP and UDP mode
		SH.ReceiveTimeout := RxTimeout;						//set receive timeout parameter
		//OS(	pHandle:= ADR(hdl),	DestHost:= Host,SDPort:= Port,DoUDP:= NOT UseTcp,res=>result ,LocalIp=>,MaxConnections := 2);
		OS(	pHandle:= ADR(hdl),	DestHost:= Host,SDPort:= Port,DoUDP:= NOT UseTcp,res=>result ,LocalIp=>,MaxConnections := 2, errState=>stateString);
		IF result = 0 THEN									//Handle was created
			Step := step + 2;			
		END_IF
		
//-------------------------------------------------
//		IF ManualClose = 1 THEN
//			Step:= 100;
//		END_IF		
//-------------------------------------------------
	
	3:	//CLIENT : wait for connection to remote
		WaitForRsp := FALSE;								//allow transmission 
		IF Host <> '' THEN 									//host address specified : connect to host
			IF UseTcp THEN	
				di := sh.CheckConnection(hdl);	
				IF di > 0 THEN								//connected	
					step := step + 3;						//go to client mode		
				END_IF
				IF di < 0 THEN								//invalid socket / timeout
					step := 100;							//go idle
					ClosedCnt := ClosedCnt + 1;
				END_IF
			ELSE			//UDP client
				SH.SetUdpHost(0,Host,Port);					//set transmit parameters manually
				step := step + 3;							//go to client mode	
			END_IF		
		ELSE												//no host specified - wait for incoming connection
			step := step + 1;								//go to server mode	
		END_IF

	4:	//SERVER : wait for connection from remote
		IF NOT Enable THEN
			step := 100;
			RETURN;
		END_IF
		IF UseTcp THEN
			wrk := SH.AcceptConnection(ListeningSocket := hdl,ADR(result));	
			IF wrk <>  SysTypes.RTS_INVALID_HANDLE THEN
				SysSockInetNtoa(ADR(SH.PartnerSck.sin_addr),partnerIp,80);	//show partner ip address
				step := step + 1;
			END_IF
			IF result = errors.ERR_SOCK_NOTSOCKET THEN	//invalid socket
				step := 1;								//start again				
			END_IF
		ELSE											//UDP server
			step := step + 1;									
			wrk := hdl;									//use same socket			
		END_IF
	
	5: //SERVER receive+respond / check listening socket (TCP only)
		IF NOT Enable THEN
			step := 100;
			RETURN;
		END_IF
		IF UseTcp THEN
			//check listening socket
			tmp := SH.AcceptConnection(ListeningSocket := hdl,ADR(result));	
			IF tmp <> SysTypes.RTS_INVALID_HANDLE THEN		//new incoming connection
				NewConnections := NewConnections + 1;
				step := 25;
				RETURN;
			END_IF
		END_IF

		IF wrk <> SysTypes.RTS_INVALID_HANDLE THEN			//connected from remote station or UDP	
			di := SH.Receive(wrk,pRxBuffer,MaxRxLen);
			
			IF di < 0 THEN									//socket has been closed/invalid socket/receive timeout
				ClosedCnt := ClosedCnt + 1;
				di := SH.Close(wrk);
				IF di > 0 THEN
					wrk := SysTypes.RTS_INVALID_HANDLE;	
					PartnerIp := '';						//no partner
					IF UseTcp THEN
						step := 4;							//go waiting for new incoming connection
					ELSE
						step := 1;							//start again							
					END_IF
				END_IF	
				RETURN;			
			END_IF
			IF di > 0 THEN									//rx data available
				RxCnt := RxCnt + 1;	
				SysSockInetNtoa(ADR(SH.PartnerSck.sin_addr),partnerIp,80);	//show partner ip address			
				SH.SetUdpHost(ADR(SH.PartnerSck),'',0);		//respond to last received partner always
				cnt := SH.Transmit(wrk,pTxBuffer,TxLen);
				IF cnt > 0 THEN
					TxCnt := TxCnt + 1;
				END_IF					
			END_IF		
		END_IF

		
		
	6: //CLIENT : transmit+get response if available 
		IF NOT Enable THEN
			step := 100;
			RETURN;
		END_IF
		IF NOT WaitForRsp THEN			
			di := SH.Transmit(hdl,pTxBuffer,TxLen);
			IF di < 0 THEN								//socket has been closed/illegal socket
				ClosedCnt := ClosedCnt + 1;
				step := 100;
				RETURN;
			END_IF
			IF di > 0 THEN								//transmission successful
				Tout(IN := FALSE, PT := T#100MS);		//restart timer
				WaitForRsp := TRUE;
				TxCnt := TxCnt + 1;						//count only really transmitted packets
			END_IF
		ELSE
			Tout(IN := TRUE);							//run timer
			cnt := SH.Receive(hdl,pRxBuffer,MaxRxLen);
			IF cnt > 0 THEN
				WaitForRsp := FALSE;
				RxCnt := RxCnt + 1;
			ELSIF cnt < 0 THEN					
				ClosedCnt := ClosedCnt + 1;
				step := 100;
				RETURN;				
			ELSE
				IF Tout.Q THEN
					TimeoutCnt := TimeoutCnt + 1;				
					WaitForRsp := FALSE;
				END_IF
			END_IF			
		END_IF


	25:		//close additional incoming connection
		di := SH.Close(tmp);
		IF di > 0 THEN
			step := step - 20;			//go back
		END_IF


	100:	//close main socket
	
//-------------------------------------------------
//		IF ManualClose = 1 THEN
//			ManualClose := 0;
//		END_IF		
//-------------------------------------------------	

	  PartnerIp := '';									//no partner
	  IF hdl <> SysTypes.RTS_INVALID_HANDLE THEN	
		di := SH.Close(hdl);
		IF di > 0 THEN
			hdl := SysTypes.RTS_INVALID_HANDLE;	
			step := step + 1;
		END_IF
	  ELSE
		step := step + 1;
	  END_IF
	  
	101:	//close tcp working socket
	  IF wrk <> SysTypes.RTS_INVALID_HANDLE THEN	
		di := SH.Close(wrk);
		IF di > 0 THEN
			wrk := SysTypes.RTS_INVALID_HANDLE;	
			step := 0;
		END_IF
	  ELSE
		step := 0;
	  END_IF

		
	200: //error 
		IF NOT Enable THEN
			step := 0;
			RETURN;
		END_IF	


END_CASE

END_FUNCTION_BLOCK

// Device/Application/Gateway/SampleReadDriveParameter
PROGRAM SampleReadDriveParameter //reads parameter from inverter 
//set bSendRequest:=TRUE to enable operation
VAR
	setcomIEC: SetCom_IEC_Slave := //setcom instance
	(
		bEnable:= TRUE, 
		iTargetNode:=0 , 
		iTargetAddress:=16#0200,	//e.g. inverter exeption state, 
		iService:=14, //can open compatible service
		bySet:=0 , //set 0
		bWriteActive:=FALSE, //read parameter
		byMaxInverterBusyCnt:=5 , 
		byMaxTimeOutCnt:=5 , 
		timSendInterval:=T#100MS
	);		
END_VAR

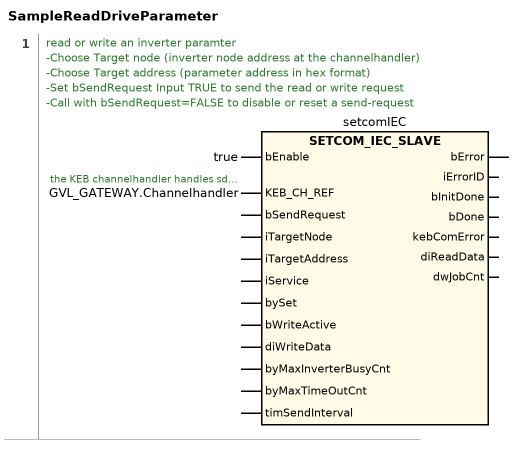
// NETWORK 1
// read or write an inverter paramter
//
// -Choose Target node (inverter node address at the channelhandler)
// -Choose Target address (parameter address in hex format)
// -Set bSendRequest Input TRUE to send the read or write request
// -Call with bSendRequest=FALSE to disable or reset a send-request
//   GVL_GATEWAY.Channelhandler: the KEB channelhandler handles sdo communication to keb drives
setcomIEC(bEnable := true, KEB_CH_REF := GVL_GATEWAY.Channelhandler); // SETCOM_IEC_SLAVE

END_PROGRAM

// Device/Application/Gateway/SampleReadMultipleParameter
(*This sample shows how to read multiple parameters with one instance of the IecSlave*)
PROGRAM SampleReadMultipleParameter


VAR CONSTANT
	LAST_INDEX:BYTE:= 2;(*Enter number of parameters to read - 1 (array goes from 0 to LAST_INDEX)*)
	PARA_ADDRESS:ARRAY [0..LAST_INDEX] OF INT:= (*Enter parameter addresses for reading*)
	[
		16#0001,//address 1
		16#0002,//address 2
		16#0003//address 3
	]; 

END_VAR

VAR_INPUT
	TargetNode:INT:=0; //inverter node 
	Reset:BOOL;		//Reset error
END_VAR

VAR_OUTPUT
	ErrorID:eSetComError;	//error id
	ComError:KebComErrors;	//com error id
	Error:BOOL;	//error during reading
	Done:BOOL;	//reading finished
END_VAR
VAR
	IecSlave: SetCom_IEC_Slave;
	ReadData:ARRAY [0..LAST_INDEX] OF DINT; (*Parameter values will be copied to this array*)
	State:INT;
	i:INT;	//loop counter
	ResetOld:BOOL;
END_VAR

CASE State OF //statemachine
	
	0:	//set send options
	//=================================================================================================
		IecSlave.iTargetNode:=TargetNode; 
		IecSlave.iService:=14;	//can open compatible service
		IecSlave.bySet:=0;	
		IecSlave.bEnable:=TRUE; //enables communication interface, do not disable!
		IecSlave.byMaxInverterBusyCnt:=5; //max. retry cnt when inverter busy
		IecSlave.byMaxTimeOutCnt:=5;		//max. retry cnt when timeout occured
		IecSlave.bWriteActive:=FALSE; //read access
		
		IecSlave(KEB_CH_REF:= GVL_GATEWAY.Channelhandler, bSendRequest:= FALSE);
		
		//reset status
		ErrorID:=0;
		ComError:=0;
		Error:=FALSE;
		Done:=FALSE;
		i:=0;
		
		State:=1;//goto next step
		
	1://send request
	//=================================================================================================
		//read all parameters and save into data array
		IecSlave 
		(
			KEB_CH_REF:=GVL_GATEWAY.ChannelHandler,
			bSendRequest:=TRUE, 
			bWriteActive:=FALSE, 
			iTargetAddress := PARA_ADDRESS[i]
		);
		
		IF IecSlave.bError THEN
			ErrorID:=IecSlave.iErrorID;
			ComError:=IecSlave.kebComError;
			Error:=TRUE;
			State:=-1;
		ELSIF IecSlave.bDone THEN
			ReadData[i]:=IecSlave.diReadData;
			IecSlave(KEB_CH_REF:=GVL_GATEWAY.ChannelHandler,bSendRequest:=FALSE); //reset FB
			ErrorID:=0;
			ComError:=0;
			Error:=FALSE;
			Done:=TRUE;	
			i:=i+1 ;	//count up and continue with next address
			IF i > LAST_INDEX THEN  (*all parameters done-->next state*)
				i:=0;
				State:=2;
			END_IF
		END_IF
			
	
	2: 	//reading finished
		IF Reset AND NOT ResetOld THEN
			State:=0;
		END_IF
		//optional do again: //State:=-2;
	
	-1://error: sending failed--> toDo: errorhandling
		IF Reset AND NOT ResetOld THEN
			State:=0;
		END_IF
	
END_CASE
ResetOld:=Reset; //edge detection

END_PROGRAM

// Device/Application/Gateway/SampleWriteDriveParameter
PROGRAM SampleWriteDriveParameter
VAR
	IecSlave: SetCom_IEC_Slave;
	State: INT;
	diWriteData: DINT:=1; //data to write into inverter address
	iErrorID: eSetComError;
	comError: KebComErrors;
END_VAR


	
	CASE State OF //statemachine
		
		0:	//set send options
			IecSlave.iTargetNode:= 0; 			//inverter at node 0
			IecSlave.iService :=14;	//can open compatible service
			IecSlave.bySet :=0;	
			IecSlave.bEnable:=TRUE ; //enables communication interface, do not disable!
			IecSlave.iTargetAddress := 16#0A20;	//inverter analog out setting (an32);
			IecSlave.byMaxInverterBusyCnt :=10; //max. retry cnt when inverter busy
			IecSlave.byMaxTimeOutCnt := 5;		//max. retry cnt when timeout occured
			IecSlave.bWriteActive := TRUE; //enable writing
			
			State:=State+1;//goto next step
			
			//IecSlave.timSendInterval := T#100MS;//optional send interval for cyclic writing
		
		1://send request

			IecSlave(
				KEB_CH_REF:= GVL_GATEWAY.Channelhandler, 	
				bSendRequest:= TRUE, //start send request
				diWriteData:= diWriteData); 
			
			//check functionblock feedback
			IF IecSlave.bDone THEN //done				
				IF IecSlave.bError THEN //done with error
					//keep last error
					iErrorID := IecSlave.iErrorID;
					comError := IecSlave.kebComError;
					//optional:call with bSendRequest=false to reset fb
						//IecSlave(KEB_CH_REF:= GVL_GATEWAY.Channelhandler, bSendRequest:= FALSE);
					State:=-1;//goto error state
				ELSE	//sucessfully done
					IecSlave(KEB_CH_REF:= GVL_GATEWAY.Channelhandler, bSendRequest:= FALSE); //call with bSendRequest=false to reset fb
					iErrorID:=0;
					comError:=0;
					State:=2;	//goto next state	
				END_IF	
			END_IF	
		
		2: 	//writing finished
					
			//optional do again: State:= 1; 
			
			
		-1://error: sending failed--> toDo: errorhandling
			IecSlave(KEB_CH_REF:= GVL_GATEWAY.Channelhandler); //, bSendRequest:= FALSE);
	
	END_CASE

END_PROGRAM

// Device/Application/SDO_RW/FB/ReadPara
FUNCTION_BLOCK ReadPara
VAR_INPUT
	StartReading: BOOL;			//TRUE 		на время чтения
	ContinuousReading: BOOL;	//TRUE 		чтобы постоянно шло чтение параметра
	SlaveAddr: UINT;			//KEB_F5_generic_MDP_.PhysSlaveAddr		(похоже - это адрес EtherCAT)
	Index: WORD;				//16#2236			адрес параметра с прибавлением 2000. В этом примере это ru.54)
	SubIndex: BYTE;				//16#1				субиндекс (вроде бы везде 1)
	ReadInterval: DINT;			//200				в КЕБе ставят 200мс
END_VAR
VAR_OUTPUT
	Value: DINT;
	Done: BOOL;
END_VAR
VAR
	EC_COE_Read:  ETC_CO_SdoRead4;
	Busy, Reading_Err: BOOL;
	Execute: BOOL;
	Busy_Fall: F_TRIG;
	Reading_Step: INT;
	Value_internal: ARRAY [1..4] OF BYTE; 
	T_Out: TON;
	ReadIntervalTimer: TON;
	//Val: DINT;
	//nnn: DINT;
	mmm: DINT;
END_VAR

IF StartReading THEN
CASE Reading_Step OF
	0://Init
	
	EC_COE_Read.usiCom:= 1; 
	EC_COE_Read.uiDevice:= SlaveAddr;  
	EC_COE_Read.wIndex:= Index; 
	EC_COE_Read.bySubindex:= SubIndex; 
	EC_COE_Read.udiTimeOut:= 1000; 
	//EC_COE_Read(xExecute:= FALSE, xAbort := FALSE);
	Reading_Step := Reading_Step + 1; 
	
	1://Call untill falling edge bBusy or bError
		EC_COE_Read(xExecute:= TRUE,xAbort := FALSE, abyData => Value_internal); 
	
		//Watchdog timer	
		IF NOT Done THEN
			T_Out(IN:= TRUE, PT:= T#500MS);
		END_IF;
			
		IF EC_COE_Read.xDone AND NOT EC_COE_Read.xError THEN//Copy data to output value
			Done := TRUE;
			//mmm := mmm + 1;
			Value_internal := EC_COE_Read.abyData; 
			Value := DWORD_TO_DINT(ArrayOfByte_to_Dword(Data := Value_Internal));
			T_Out(IN:= FALSE, PT:= T#500MS);//Reset watchdog
		END_IF
		
		IF EC_COE_Read.xError OR T_Out.Q THEN//In case of watchdog or error go to reset
			Reading_Step := 2;
			T_Out(IN:= FALSE, PT:= T#500MS);
		END_IF;

		ReadIntervalTimer(IN:= ContinuousReading, PT:= DINT_TO_TIME(ReadInterval));
		IF ContinuousReading AND ReadIntervalTimer.Q THEN//reading was succesfull, after reading pause go to reset
			ReadIntervalTimer(IN:= FALSE, PT:= DINT_TO_TIME(ReadInterval));
			Reading_Step := 2;
		END_IF; 
		
	2://Reset FB
		
			EC_COE_Read(xExecute:= FALSE, xAbort := TRUE);
			Done := FALSE;
			Reading_Step := 0;
		
END_CASE
ELSE
	EC_COE_Read(xExecute:= FALSE, xAbort := FALSE);
	Done := FALSE;
	Reading_Step := 0;
END_IF

END_FUNCTION_BLOCK

// Device/Application/SDO_RW/FB/WritePara
FUNCTION_BLOCK WritePara
VAR_INPUT
	StartWriting: BOOL;
	SlaveAddr: UINT;
	Index: WORD;
	SubIndex: BYTE;
	Value: DINT;
	DataLength: USINT;
END_VAR
VAR_OUTPUT
	
	Done: BOOL;
END_VAR
VAR
	EC_COE_Write:  ETC_CO_SdoWrite4;
	Busy, Reading_Err: BOOL;
	Execute: BOOL;
	Busy_Fall: F_TRIG;
	Reading_Step: INT;
	Value_internal: ARRAY [1..4] OF BYTE; 
	T_Out: TON;
	ReadIntervalTimer: TON;
	//Val: DINT;
	//nnn: DINT;
	mmm: DINT;
END_VAR

IF StartWriting THEN
CASE Reading_Step OF
	0://Init
	
	 
	EC_COE_Write.usiCom:= 1; 
	EC_COE_Write.uiDevice:= SlaveAddr;  
	EC_COE_Write.wIndex:= Index; 
	EC_COE_Write.bySubindex:= SubIndex; 
	EC_COE_Write.udiTimeOut:= 1000; 
	//EC_COE_Write(xExecute:= FALSE, xAbort := FALSE);
	Reading_Step := Reading_Step + 1;
	EC_COE_Write.usiDataLength := DataLength;
	Dint_ToArrayOfByte(); 
	
	1://Call untill falling edge bBusy or bError
	
		IF NOT Done THEN
			EC_COE_Write(xExecute:= TRUE, xAbort := FALSE,abyData := Value_internal); 
		END_IF;
		
		//Watchdog timer	
		//IF NOT Done THEN
			//T_Out(IN:= TRUE, PT:= T#1S);
		//END_IF;
			
		IF EC_COE_Write.xDone AND NOT EC_COE_Write.xError THEN//Copy data to output value
			Done := TRUE;
			T_Out(IN:= FALSE, PT:= T#500MS);//Reset watchdog
		END_IF
		
		IF EC_COE_Write.xError OR T_Out.Q THEN//In case of watchdog or error go to reset
			Reading_Step := 2;
			T_Out(IN:= FALSE, PT:= T#500MS);
		END_IF;

	2://Reset FB
		
			EC_COE_Write(xExecute:= FALSE, xAbort := TRUE);
			Done := FALSE;
			Reading_Step := 0;
		
END_CASE
ELSE
	EC_COE_Write(xExecute:= FALSE, xAbort := FALSE);
	Done := FALSE;
	Reading_Step := 0;
END_IF

ACTION Dint_ToArrayOfByte:
Value_internal[1] := DWORD_TO_BYTE(DINT_TO_DWORD(Value));
Value_internal[2] := DWORD_TO_BYTE(SHR(DINT_TO_DWORD(Value), 8));
Value_internal[3] := DWORD_TO_BYTE(SHR(DINT_TO_DWORD(Value), 16));
Value_internal[4] := DWORD_TO_BYTE(SHR(DINT_TO_DWORD(Value), 24));
END_ACTION

END_FUNCTION_BLOCK
